(* PLC project PLC, Beckhoff Automation GmbH TwinCAT PLC Control 3.5.13.20 *)
(* stored: creationDateTime 2021-09-02T10:04:16.8056045, modificationDateTime 2021-09-02T10:04:16.8120124 *)

(*-----------------------------------------版本信息-----------------------------------------
第一版本：		V1.0.0
功能说明：		边缘触发功能块集合
开发者：		Long.Yun
开发时间：		2021.09.02

变更版本：
版本			变更者		变更时间		变更说明
------------------------------------------------------------------------------------------*)
FUNCTION_BLOCK BFB_Trigger
VAR_INPUT
	//触发位
	bIn			:BOOL;
END_VAR

VAR_OUTPUT
	//边沿交替输出
	bTrig		:BOOL;
	//上升沿输出
	bRiseTrig	:BOOL;
	//下降沿输出
	bFallTrig	:BOOL;
END_VAR

VAR
	{attribute 'hide'}
	fbTrigR		:R_TRIG;
	{attribute 'hide'}
	fbTrigF		:F_TRIG;
END_VAR

            fbTrigR(CLK := bIn, Q =>bRiseTrig);

fbTrigF(CLK := bIn, Q => bFallTrig);

bTrig := bRiseTrig OR bFallTrig;
          
END_FUNCTION_BLOCK
